FUNCTION_BLOCK HAL_DI_Channel IMPLEMENTS I_HAL_DI
VAR_INPUT
	terminal_address		: WORD;
END_VAR
VAR_OUTPUT
END_VAR
VAR
	_errId:UINT;
	_xValue: BOOL;
	_channel_number: UINT;
END_VAR

PROPERTY errId : UINT
GET
errId := _errId;
END_GET
END_PROPERTY

METHOD FB_init : BOOL
VAR_INPUT
	bInitRetains 	: BOOL; // if TRUE, the retain variables are initialized (warm start / cold start)
	bInCopyCode 	: BOOL;  // if TRUE, the instance afterwards gets moved into the copy code (online change)
    channel_number  : UINT;
END_VAR

_channel_number :=channel_number;
END_METHOD

PROPERTY terminal_value : bool
SET
_xValue:=terminal_value;
END_SET
END_PROPERTY

PROPERTY WcState : bool
GET
END_GET
SET
END_SET
END_PROPERTY

{warning 'add property implementation'}
PROPERTY xValue : BOOL
GET
xValue:=_xValue;
END_GET
END_PROPERTY

END_FUNCTION_BLOCK

(* stored: Version 1.1.0.1, ProductVersion 3.1.4024.6
   POU HAL_DI_Channel: Id {b1d1af24-c998-05f1-3746-9bdeae67a77b}, SpecialFunc None
   Folder HAL: Id {3ba1257c-608d-096a-037f-ba20c8a64160}
   Folder IO: Id {494853d3-a77f-0b99-1d9d-50b529669bb4}
   Property errId: Id {4dcbf7f9-a5dd-019a-24f5-c34e969e268c}
   Get Get: Id {07864ee9-bfc1-0814-06ce-68b0256df53d}
   Method FB_init: Id {13a93988-853b-0f7e-17ed-a973216b4a06}
   Property terminal_value: Id {0e7cab75-3369-0048-0aef-636f6b3285a2}
   Set Set: Id {975877ec-8fc6-0b96-29e7-8e4feb8aac1d}
   Property WcState: Id {d052cbf9-1a59-0912-3d51-e7a7c12cb554}
   Get Get: Id {696f6250-c2ce-0e6d-2406-1d7e8d2feab6}
   Set Set: Id {4e9daffa-df3e-0abd-0de1-ad207a16b216}
   Property xValue: Id {1c7b2364-c8f4-0977-1a1d-255b9df12e97}
   Get Get: Id {8dd4c25e-ae41-06ad-2032-a74ae88739f7} *)
